PROGRAM P_Modes

VAR
	fbRunning : FB_Running;
END_VAR

// Runs FB with given values
fbRunning(
	bAuto := G_Inputs.bAuto, 			// Auto mode controller
	bManual := G_Inputs.bManual, 		// Manual mode controller
	bStart := G_Inputs.bStartButton,	// Start button
	bStop := G_Inputs.bStopButton, 		// Stop button
	
	// Values from FB sent to GVL
	bRunning => G_Mode.bRunning,
	bRunning => G_Output.bRunning,
	bManualMode => G_Mode.bManual,
	bAutoMode => G_Mode.bAuto
);

END_PROGRAM

(* stored: Version 1.1.0.1
   POU P_Modes: Id {022044ba-8743-45e6-a82b-2e81f0455edb}, SpecialFunc None *)
